FUNCTION_BLOCK RemoveAllMover_TestSuite
VAR
	ThisTestSuite : TestSuite<TestSuiteParameter.MaxTestCount>('C:\ProgramData\Beckhoff\TwinCAT\3.1\Boot\RemoveAll_Tests.xml') := (TestSuiteName := 'RemoveAll Test Suite');
END_VAR

TaskAcceptsRemoveCommand_Test();
TaskRejectsDuplicateCommand_Test();
TaskRejectsCyclicWithNoGroup_Test();
TaskRejectsInvalidCAGroup();
TaskRejectsRemoveAllWithNoGroup_Test();

METHOD TaskAcceptsRemoveCommand_Test
VAR
	stubGroup : CollisionGroup;
	testRemoveAll : RemoveAllMoverFromGroup := (MyCollisionGroup := stubGroup);
	Expected : BOOL := TRUE;
	Actual	 : BOOL;
END_VAR
IF ThisTestSuite.Test(__POUNAME()).ExecuteTest() THEN
	Actual := SUCCEEDED(testRemoveAll.RemoveAllMover());
	ThisTestSuite.Test(__POUNAME()).AssertEqual(Expected, Actual);
END_IF
END_METHOD

METHOD TaskRejectsCyclicWithNoGroup_Test : BOOL
VAR
	stubGroup : CollisionGroup;
	testRemoveAll : RemoveAllMoverFromGroup := (MyCollisionGroup := stubGroup);
	Expected : BOOL := TRUE;
	Actual	 : BOOL;
END_VAR
IF ThisTestSuite.Test(__POUNAME()).ExecuteTest() THEN
	Actual := FAILED(testRemoveAll.Cycle());
	ThisTestSuite.Test(__POUNAME()).AssertEqual(Expected, Actual);
END_IF
END_METHOD

METHOD TaskRejectsDuplicateCommand_Test
VAR
	stubGroup : CollisionGroup;
	testRemoveAll : RemoveAllMoverFromGroup := (MyCollisionGroup := stubGroup);
	Expected : BOOL := TRUE;
	Actual	 : BOOL;
END_VAR
IF ThisTestSuite.Test(__POUNAME()).ExecuteTest() THEN
	testRemoveAll.RemoveAllMover();
	Actual := FAILED(testRemoveAll.RemoveAllMover());
	ThisTestSuite.Test(__POUNAME()).AssertEqual(Expected, Actual);
END_IF
END_METHOD

METHOD TaskRejectsInvalidCAGroup
VAR
	stubGroup : CollisionGroup;
	iStubCAGRoup : I_CollisionGroup := stubGroup;
	testRemoveAll : RemoveAllMoverFromGroup := (MyCollisionGroup := stubGroup);
	Expected : BOOL := TRUE;
	Actual	 : BOOL;
END_VAR
IF ThisTestSuite.Test(__POUNAME()).ExecuteTest() THEN
	testRemoveAll.MyCollisionGroup := 16#0;
	Actual := testRemoveAll.MyCollisionGroup = iStubCAGroup;
	ThisTestSuite.Test(__POUNAME()).AssertEqual(Expected, Actual);
END_IF
END_METHOD

METHOD TaskRejectsRemoveAllWithNoGroup_Test
VAR
	testRemoveAll : RemoveAllMoverFromGroup ;
	Expected : BOOL := TRUE;
	Actual	 : BOOL;
END_VAR
IF ThisTestSuite.Test(__POUNAME()).ExecuteTest() THEN
	Actual := FAILED(testRemoveAll.RemoveAllMover());
	ThisTestSuite.Test(__POUNAME()).AssertEqual(Expected, Actual);
END_IF
END_METHOD

END_FUNCTION_BLOCK

(* stored: Version 1.1.0.1
   POU RemoveAllMover_TestSuite: Id {eeedca17-e20e-45f9-84f5-4809781a4cf4}, SpecialFunc None
   Method TaskAcceptsRemoveCommand_Test: Id {2cfd4574-9937-4592-b537-84fc1b0143b7}
   Method TaskRejectsCyclicWithNoGroup_Test: Id {eb085bbf-96a4-47f3-90b3-c371a73f522c}
   Method TaskRejectsDuplicateCommand_Test: Id {915ffafe-cf86-4fb1-bd7f-804ac745cb61}
   Method TaskRejectsInvalidCAGroup: Id {9e44dde0-69a2-4313-9725-298644851780}
   Method TaskRejectsRemoveAllWithNoGroup_Test: Id {ebe2e133-0037-473a-a8bc-09016778cc0e} *)
